(*
SPDX-FileCopyrightText: © 2026 Oleksandr Tiutyk <trofimich@gmail.com>
SPDX-License-Identifier: MIT
License: https://opensource.org/license/mit
*)

(*!
<summary>Stores an ordered sequence of generic values with fixed or dynamic capacity.</summary>
<description>
CreateEnumerator allocates an independent cursor owned by its caller. The collection must remain alive while
that cursor is used. Dynamic growth preserves the existing buffer on allocation failure and invokes the
terminal allocation-failure mechanism. Sort uses GENERIC_VALUE.CompareTo unless an explicit borrowed comparer
is supplied; descriptors preserve OBJECT and USER_DEFINED categories. Successful insertion transfers disposal
responsibility for owned payload; borrowed payload must remain alive while stored. The caller-side descriptor
copy is not reset and must not be released again after transfer. Independent owning aliases and overlapping
owned allocations are unsupported. Entries retain order and duplicates. Same-allocation replacement preserves
ownership without releasing retained storage. Get, FindSingle and enumerators only borrow payload.
ContainsGeneric defaults to releasing its query. Validators are borrowed for the collection lifetime. No
locking or mutation-version checks are implemented; callbacks that mutate the collection can invalidate
in-progress operations. Generic lookup with requested query release also attempts cleanup on lookup failure
before propagating the captured exception; terminal OOM takes precedence.
Instances cannot be assigned by value: copying backing pointers or disposal responsibility would create
unsafe aliases. Interface references still borrow this instance; copying an interface does not clone storage.
</description>
*)

{attribute 'no_explicit_call' := 'do not call this function block directly'}
FUNCTION_BLOCK List 
VAR_GENERIC CONSTANT
 	{attribute 'hide'} 
	//! <summary>Inline capacity; zero selects dynamic backing storage.</summary>
	_StaticCapacity : TOF_Core.DINT_LENGTH := 0;
END_VAR
EXTENDS TOF_Core.Object IMPLEMENTS IList
VAR_INPUT
	//! <summary>Number of slots added when dynamic storage is full; must be positive when growth is required.</summary>
	DefaultDynamicAllocationElementCount : BYTE := 10;	
END_VAR
VAR_STAT
	//! <summary>Class name shared by all instances of this function block.</summary>
	{attribute 'hide'} 
	_ClassName : STRING := __POUNAME();
END_VAR
VAR
	{attribute 'hide'} 
	_ValueValidator : TOF_Core.IGenericValueValidator;

	{attribute 'hide'} 
	_Array : POINTER TO TOF_Core.GENERIC_VALUE;
	{attribute 'hide'} 
	_StaticArray : ARRAY [0.._StaticCapacity - 1] OF TOF_Core.GENERIC_VALUE;
	
	{attribute 'hide'} 
	_DynamicCapacity : TOF_Core.DINT_LENGTH;
	{attribute 'hide'} 
	_Length : TOF_Core.DINT_LENGTH;
END_VAR

(*!
<summary>Grows the dynamic element buffer while preserving existing values.</summary>
<description>
Static instances return without allocation. A positive increment must fit DINT capacity and the UDINT
allocation-byte limit; invalid ranges raise ArgumentOutOfRangeException before storage changes. A null
allocation invokes the terminal allocation-failure mechanism before copying or deleting the old buffer.
Existing descriptors are moved without cloning payload; incoming ownership is not accepted by this helper.
Descendants cannot override this storage operation; capacity, indexing and disposal remain governed by this
collection implementation.
</description>
*)
METHOD PROTECTED FINAL AllocateMemory 
VAR_INPUT
	elementCount : TOF_Core.DINT_LENGTH;
END_VAR
VAR CONSTANT
	//! <summary>Bytes per capacity slot, including descriptor storage and any hash-index arrays.</summary>
	ENTRY_ALLOCATION_SIZE : ULINT := XSIZEOF(TOF_Core.GENERIC_VALUE);
END_VAR
VAR
	newMemory : POINTER TO TOF_Core.GENERIC_VALUE;
	newCapacity : ULINT;

END_VAR
IF NOT Dynamic THEN
	RETURN;
END_IF

IF elementCount <= TOF_Core.SignedInt32.ZERO THEN
	TOF_Core.Exceptions.ThrowArgumentOutOfRange(
		sourceNamespaceName := NamespaceName,
		sourceClassName := ClassName,
		sourcePOUName := __POUNAME(),
		sourcePosition := __POSITION(),
		argumentName := 'elementCount',
		argumentValue := elementCount
	);
END_IF

newCapacity := TO_ULINT(_DynamicCapacity) + TO_ULINT(elementCount);

IF newCapacity > TO_ULINT(TOF_Core.SignedInt32.MAX_VALUE)
	OR_ELSE newCapacity > TO_ULINT(TOF_Core.UnsignedInt32.MAX_VALUE) / ENTRY_ALLOCATION_SIZE
THEN
	TOF_Core.Exceptions.ThrowArgumentOutOfRange(
		sourceNamespaceName := NamespaceName,
		sourceClassName := ClassName,
		sourcePOUName := __POUNAME(),
		sourcePosition := __POSITION(),
		argumentName := 'capacity',
		argumentValue := newCapacity
	);
END_IF

newMemory := __NEW(BYTE, TO_UDINT(ENTRY_ALLOCATION_SIZE * newCapacity));

IF newMemory = 0 THEN
	TOF_Core.DynamicMemoryManager.RaiseAllocationFailure();
END_IF

IF _Length > TOF_Core.SignedInt32.ZERO THEN
	Tc2_System.MEMCPY(destAddr := newMemory, srcAddr := _Array, n := TO_UDINT(ENTRY_ALLOCATION_SIZE * TO_ULINT(_Length)));
END_IF

IF _Array <> 0 THEN
	__DELETE(_Array);
END_IF

_DynamicCapacity := TO_DINT(newCapacity);
_Array := newMemory;
END_METHOD

(*!
<summary>Copies a value and appends the owned descriptor.</summary>
<description>
Borrows the original during the call. isObject = TRUE requires a live Object FB instance implementing
ICloneable; other data is copied as bytes without recursively cloning references. A prepared copy is released
if insertion fails before acceptance; exceptions propagate. Engine-managed exception objects are unsupported.
index is meaningful only on success. Descendants cannot override this storage operation; capacity, indexing
and disposal remain governed by this collection implementation.
The original failure is captured before cleanup so nested cleanup handling cannot replace its payload.
A static native wrapper is cloned before cleanup; failure to capture still attempts prepared-copy disposal.
Terminal allocation failure takes precedence and no exception clone is allocated after its latch is set.
</description>
*)
METHOD FINAL AppendCopy : IList
VAR_INPUT
	value : ANY;
	isObject : BOOL := FALSE;
END_VAR
VAR_OUTPUT
	index : TOF_Core.DINT_INDEX;
END_VAR
VAR
	exceptionCode : __SYSTEM.ExceptionCode;
	caughtException : TOF_Core.IException;
	genericValue : TOF_Core.GENERIC_VALUE;
END_VAR

genericValue := TOF_Core.GenericValueFactory.FromAnyType(
		value := value,
		isObject := isObject,
		memoryManagementBehavior := TOF_Core.GENERIC_MEMORY_MANAGEMENT_BEHAVIOR.CLONE_ORIGINAL_VALUE_AND_OWNS_MEMORY
	);

__TRY
	AppendCopy := AppendGeneric(value := genericValue, index => index);
__CATCH(exceptionCode)
	caughtException := TOF_Core.ExceptionManager.GetLastException(
		exceptionCode := exceptionCode,
		catchPointNamespaceName := NamespaceName,
		catchPointPOUName := __POUNAME(),
		catchPointPosition := __POSITION()
	);
__ENDTRY

IF caughtException <> 0 THEN
	__TRY
		TOF_Core.DynamicMemoryManager.RaiseIfAllocationFailed();

		IF NOT caughtException.IsDynamicInstance THEN
			__QUERYINTERFACE(caughtException.Clone(), caughtException);
		END_IF
	__CATCH(exceptionCode)
		genericValue.Release();

		TOF_Core.ExceptionManager.ReThrowLastException(
			exceptionCode := exceptionCode,
			catchPointNamespaceName := NamespaceName,
			catchPointPOUName := __POUNAME(),
			catchPointPosition := __POSITION()
		);
	__ENDTRY

	genericValue.Release();

	TOF_Core.ExceptionManager.Throw(exception := caughtException);
END_IF
END_METHOD

(*!
<summary>Appends a descriptor to the list.</summary>
<description>
Successful insertion transfers disposal responsibility for owned payload; borrowed payload must remain alive
while stored. The caller-side descriptor copy is not reset and must not be released again after transfer.
Independent owning aliases and overlapping owned allocations are unsupported. Delegates to InsertGeneric;
index is meaningful only on success. Descendants cannot override this storage operation; capacity, indexing
and disposal remain governed by this collection implementation.
</description>
*)
METHOD FINAL AppendGeneric : IList
VAR_INPUT
	value : TOF_Core.GENERIC_VALUE;
END_VAR
VAR_OUTPUT
	index : TOF_Core.DINT_INDEX;
END_VAR
index := _Length;

AppendGeneric := InsertGeneric(index := index, value := value);
END_METHOD

(*!
<summary>Reports the currently allocated number of slots.</summary>
<description>
Units are bytes for ByteList and entries for other collections. Static capacity is fixed; dynamic capacity can
change on growth or clearing. This is not a guarantee that the next allocation succeeds.
</description>
*)
{attribute 'monitoring' := 'call'}
PROPERTY FINAL Capacity : TOF_Core.DINT_LENGTH
GET
Capacity := SEL(_StaticCapacity = 0, _StaticCapacity, _DynamicCapacity);
END_GET
END_PROPERTY

(*!
<summary>Borrows the concrete collection class name without transferring storage ownership.</summary>
*)
{attribute 'monitoring' := 'call'}
PROPERTY ClassName : REFERENCE TO STRING
GET
ClassName REF= _ClassName;
END_GET
END_PROPERTY

(*!
<summary>Removes all entries and releases dynamic backing storage.</summary>
<description>
Owned payload is released best effort through GENERIC_VALUE.Release; borrowed storage is not freed. Static
capacity and the borrowed validator are retained. Dynamic capacity becomes zero. Returns this collection and
invalidates positions and views. Cleanup callbacks must not reenter mutation. Descendants cannot override this
storage operation; capacity, indexing and disposal remain governed by this collection implementation.
</description>
*)
METHOD FINAL Clear : IList
VAR
	i : DINT;
END_VAR
Clear := THIS^;

FOR i := 0 TO _Length - 1 DO
	_Array[i].Release();						
END_FOR	

_Length := 0;
_DynamicCapacity := 0;

IF _Array <> 0 AND_THEN Dynamic THEN
	__DELETE(_Array);	
END_IF
END_METHOD

(*!
<summary>Searches for a value using default generic equality.</summary>
<description>
Borrows the ANY argument during a linear search without cloning or releasing it. isObject = TRUE means a live
Object FB instance, not a pointer or interface variable. Equality exceptions propagate; callbacks that mutate
the collection can invalidate traversal. Descendants cannot override this storage operation; capacity,
indexing and disposal remain governed by this collection implementation.
</description>
*)
METHOD FINAL Contains : BOOL
VAR_INPUT
	value : ANY;
	isObject : BOOL := FALSE;
END_VAR
VAR
	genericValue : TOF_Core.GENERIC_VALUE;
	i : TOF_Core.DINT_INDEX;
END_VAR

genericValue := TOF_Core.GenericValueFactory.FromAnyType(
		value := value,
		isObject := isObject,
		memoryManagementBehavior := TOF_Core.GENERIC_MEMORY_MANAGEMENT_BEHAVIOR.STORE_ORIGINAL_REFERENCE_AND_NOT_OWNS_MEMORY
	);

FOR i := 0 TO _Length - 1 DO
	IF _Array[i].Equals(otherValue := genericValue) THEN
		Contains := TRUE;
		RETURN;
	END_IF
END_FOR
END_METHOD

(*!
<summary>Searches for an equal generic value and optionally releases the query.</summary>
<description>
Uses GENERIC_VALUE.Equals in a linear search. releaseValue defaults to TRUE: after a completed search, Release
is called on the local query copy, including on a miss. Caller-side aliases are not reset. The query must not
own storage retained by the collection. Requested release is attempted after both successful lookup and lookup
failure. Before cleanup, the original framework exception is retained and a borrowed static system exception
is cloned to preserve its code, catch point and timestamps across cleanup callbacks. The captured exception is
then propagated through ExceptionManager.Throw in the current cyclic task; native errors use the framework
SystemException representation. If capturing the system exception fails with terminal OOM, query cleanup is
still attempted and terminal OOM takes precedence. Terminal allocation state is never cleared. Release is best
effort and does not prove successful deallocation. Cleanup callbacks must not reenter collection mutation.
Descendants cannot override this storage operation; capacity, indexing and disposal remain governed by this
collection implementation.
</description>
*)
METHOD FINAL ContainsGeneric : BOOL
VAR_INPUT
	value : TOF_Core.GENERIC_VALUE;
	releaseValue : BOOL := TRUE;
END_VAR
VAR
	exceptionCode : __SYSTEM.ExceptionCode;
	caughtException : TOF_Core.IException;

	i : DINT;
END_VAR
__TRY
	FOR i := 0 TO _Length - 1 DO
		IF _Array[i].Equals(otherValue := value) THEN
			ContainsGeneric := TRUE;
			EXIT;
		END_IF
	END_FOR
__CATCH(exceptionCode)
	caughtException := TOF_Core.ExceptionManager.GetLastException(
		exceptionCode := exceptionCode,
		catchPointNamespaceName := NamespaceName,
		catchPointPOUName := __POUNAME(),
		catchPointPosition := __POSITION()
	);
__ENDTRY

IF releaseValue THEN
	IF caughtException <> 0 AND_THEN NOT caughtException.IsDynamicInstance THEN
		__TRY
			TOF_Core.DynamicMemoryManager.RaiseIfAllocationFailed();
			__QUERYINTERFACE(caughtException.Clone(), caughtException);
		__CATCH(exceptionCode)
			value.Release();

			TOF_Core.ExceptionManager.ReThrowLastException(
				exceptionCode := exceptionCode,
				catchPointNamespaceName := NamespaceName,
				catchPointPOUName := __POUNAME(),
				catchPointPosition := __POSITION()
			);
		__ENDTRY
	END_IF

	value.Release();
END_IF

IF caughtException <> 0 THEN
	TOF_Core.ExceptionManager.Throw(exception := caughtException);
END_IF
END_METHOD

(*!
<summary>Creates an independent enumerator owned by the caller.</summary>
<description>
The caller must explicitly release the enumerator and keep this collection alive while using it. Allocation
failure invokes DynamicMemoryManager.RaiseAllocationFailure without a heap exception; it is terminal and is
not returned as a recoverable null result.
</description>
*)
METHOD CreateEnumerator : TOF_Core.IEnumerator
VAR
	enumerator : POINTER TO ListEnumerator;
END_VAR
enumerator := __NEW(ListEnumerator(list := THIS^));

IF enumerator = 0 THEN
	TOF_Core.DynamicMemoryManager.RaiseAllocationFailure();
END_IF

CreateEnumerator := enumerator^;
END_METHOD

(*!
<summary>Reports whether storage can grow dynamically.</summary>
<description>
Static capacity zero selects dynamic storage. Dynamic collections can still fail to allocate.
</description>
*)
{attribute 'monitoring' := 'call'}
PROPERTY FINAL Dynamic : BOOL
GET
Dynamic := _StaticCapacity = 0;
END_GET
END_PROPERTY

(*!
<summary>Reports whether the collection has no entries.</summary>
<description>
Reflects Length; not a check of payload lifetime or memory health.
</description>
*)
{attribute 'monitoring' := 'call'}
PROPERTY FINAL Empty : BOOL
GET
Empty := _Length <= 0;
END_GET
END_PROPERTY

(*!
<summary>Releases owned payload and backing storage during destruction.</summary>
<description>
Calls Clear; lifecycle methods and payload cleanup callbacks must not raise exceptions or reenter mutation.
Payload release is best effort, not proof of successful destruction. No separate copy-code ownership handoff
is implemented.
</description>
*)

METHOD FB_exit : BOOL
VAR_INPUT
	bInCopyCode : BOOL; 
END_VAR
Clear();
END_METHOD

(*!
<summary>Binds the optional validator and inline storage during initialization.</summary>
<description>
The validator is borrowed and must remain alive while used; it is not invoked here. Static storage is bound
without allocation. Lifecycle methods must not raise exceptions. No explicit online-change relocation repair
is implemented.
</description>
*)
METHOD FB_init : BOOL
VAR_INPUT
	bInitRetains : BOOL; // TRUE: the retain variables are initialized (reset warm / reset cold)
	bInCopyCode : BOOL; // TRUE: the instance will be copied to the copy code afterward (online change)
	valueValidator : TOF_Core.IGenericValueValidator;
END_VAR
_ValueValidator := valueValidator;

IF NOT Dynamic THEN
	_Array := ADR(_StaticArray); 
END_IF
END_METHOD

(*!
<summary>Finds a predicate match in the requested traversal direction.</summary>
<description>
skip counts matches, not visited entries. A null predicate or no match returns FALSE; outputs are meaningful
only on TRUE. The result is borrowed even if IsMemoryOwner is TRUE. Predicate input uses AsAnyType without
preserving the explicit generic OBJECT category. Predicate exceptions propagate; callbacks must not mutate the
traversed collection. Descendants cannot override this storage operation; capacity, indexing and disposal
remain governed by this collection implementation.
</description>
*)
METHOD FINAL FindSingle : BOOL
VAR_INPUT
	predicate : TOF_Core.IPredicate;
	skip : UDINT := 0;
	searchDirection : TOF_Core.SEARCH_DIRECTION := TOF_Core.SEARCH_DIRECTION.FROM_BEGINNING;
END_VAR
VAR_OUTPUT
	value : TOF_Core.GENERIC_VALUE;
	index : TOF_Core.DINT_INDEX;
END_VAR
VAR
	startSearchIndex : DINT;
	maxSearchIndex : DINT;
	indexStep : DINT;
	
	i : DINT;
	
	currentValue : __SYSTEM.AnyType;

	skippedMatchCount : UDINT := 0;
END_VAR
index := 0;
	
IF TO_DINT(skip) >= _Length OR_ELSE predicate = 0 THEN
	RETURN;
END_IF

startSearchIndex := SEL(searchDirection = TOF_Core.SEARCH_DIRECTION.FROM_BEGINNING, _Length - 1, 0);
maxSearchIndex := SEL(searchDirection = TOF_Core.SEARCH_DIRECTION.FROM_BEGINNING, 0, _Length - 1);
indexStep := SEL(searchDirection = TOF_Core.SEARCH_DIRECTION.FROM_BEGINNING, -1, 1);

FOR i := startSearchIndex TO maxSearchIndex BY indexStep DO
	currentValue := _Array[i].AsAnyType();
	
	IF predicate.Check(valueToCompare := currentValue) THEN
		IF skip = skippedMatchCount THEN
			value := _Array[i];
			index := i;
			FindSingle := TRUE;
			RETURN;
		ELSE
			skippedMatchCount := skippedMatchCount + 1;
		END_IF
	END_IF
END_FOR
END_METHOD

(*!
<summary>Reports whether fixed-capacity storage has no free slot.</summary>
<description>
Dynamic collections report FALSE even when Length equals Capacity. This does not guarantee available heap
memory.
</description>
*)
{attribute 'monitoring' := 'call'}
PROPERTY FINAL Full : BOOL
GET
Full := _StaticCapacity <> 0 AND_THEN _Length >= _StaticCapacity;
END_GET
END_PROPERTY

(*!
<summary>Borrows the descriptor at a zero-based list position.</summary>
<description>
An out-of-range index raises an exception. Returned descriptors and payload are borrowed, not clones. Do not
modify descriptor metadata or release payload through this view, even when IsMemoryOwner is TRUE. Keep the
source and borrowed storage alive; mutation or destruction can invalidate the view. Descendants cannot
override this storage operation; capacity, indexing and disposal remain governed by this collection
implementation.
</description>
*)
METHOD FINAL Get : REFERENCE TO TOF_Core.GENERIC_VALUE
VAR_INPUT
	index : TOF_Core.DINT_INDEX;
END_VAR
IF index < 0 OR_ELSE index >= _Length THEN
	TOF_Core.Exceptions.ThrowArgumentOutOfRange(
		sourceNamespaceName := NamespaceName,
		sourceClassName := ClassName,
		sourcePOUName := __POUNAME(),
		sourcePosition := __POSITION(),
		argumentName := 'index',
		argumentValue := index
	);
END_IF

Get REF= _Array[index];
END_METHOD

(*!
<summary>Copies a value and inserts it at the requested position.</summary>
<description>
Borrows the original during the call. isObject = TRUE requires a live Object FB instance implementing
ICloneable; other data is copied as bytes without recursively cloning references. A prepared copy is released
if insertion fails before acceptance; exceptions propagate. Engine-managed exception objects are unsupported.
The position may range from zero through Length inclusive. Descendants cannot override this storage operation;
capacity, indexing and disposal remain governed by this collection implementation.
The original failure is captured before cleanup so nested cleanup handling cannot replace its payload.
A static native wrapper is cloned before cleanup; failure to capture still attempts prepared-copy disposal.
Terminal allocation failure takes precedence and no exception clone is allocated after its latch is set.
</description>
*)
METHOD FINAL InsertCopy : IList
VAR_INPUT
	index : TOF_Core.DINT_INDEX;
	value : ANY;
	isObject : BOOL := FALSE;
END_VAR
VAR
	exceptionCode : __SYSTEM.ExceptionCode;
	caughtException : TOF_Core.IException;
	genericValue : TOF_Core.GENERIC_VALUE;
END_VAR

genericValue := TOF_Core.GenericValueFactory.FromAnyType(
		value := value,
		isObject := isObject,
		memoryManagementBehavior := TOF_Core.GENERIC_MEMORY_MANAGEMENT_BEHAVIOR.CLONE_ORIGINAL_VALUE_AND_OWNS_MEMORY
	);

__TRY
	InsertCopy := InsertGeneric(index := index, value := genericValue);
__CATCH(exceptionCode)
	caughtException := TOF_Core.ExceptionManager.GetLastException(
		exceptionCode := exceptionCode,
		catchPointNamespaceName := NamespaceName,
		catchPointPOUName := __POUNAME(),
		catchPointPosition := __POSITION()
	);
__ENDTRY

IF caughtException <> 0 THEN
	__TRY
		TOF_Core.DynamicMemoryManager.RaiseIfAllocationFailed();

		IF NOT caughtException.IsDynamicInstance THEN
			__QUERYINTERFACE(caughtException.Clone(), caughtException);
		END_IF
	__CATCH(exceptionCode)
		genericValue.Release();

		TOF_Core.ExceptionManager.ReThrowLastException(
			exceptionCode := exceptionCode,
			catchPointNamespaceName := NamespaceName,
			catchPointPOUName := __POUNAME(),
			catchPointPosition := __POSITION()
		);
	__ENDTRY

	genericValue.Release();

	TOF_Core.ExceptionManager.Throw(exception := caughtException);
END_IF
END_METHOD

(*!
<summary>Inserts a descriptor and shifts subsequent entries to the right.</summary>
<description>
Successful insertion transfers disposal responsibility for owned payload; borrowed payload must remain alive
while stored. The caller-side descriptor copy is not reset and must not be released again after transfer.
Independent owning aliases and overlapping owned allocations are unsupported. index may range from zero
through Length inclusive. Invalid indices and full static storage raise exceptions. Validation precedes
insertion. Dynamic growth rejects nonpositive increments and unrepresentable capacity or allocation sizes
before insertion. Descendants cannot override this storage operation; capacity, indexing and disposal remain
governed by this collection implementation.
</description>
*)
METHOD FINAL InsertGeneric : IList
VAR_INPUT
	index : TOF_Core.DINT_INDEX;
	value : TOF_Core.GENERIC_VALUE;	
END_VAR
VAR
	
	i : DINT;
END_VAR
IF index < 0 OR_ELSE index > _Length THEN
	TOF_Core.Exceptions.ThrowArgumentOutOfRange(
		sourceNamespaceName := NamespaceName,
		sourceClassName := ClassName,
		sourcePOUName := __POUNAME(),
		sourcePosition := __POSITION(),
		argumentName := 'index',
		argumentValue := index
	);
END_IF

IF _ValueValidator <> 0 THEN
	_ValueValidator.Validate(validatedObjectName := GetName(), valueToValidate := value);
END_IF

InsertGeneric := THIS^;

IF _Length >= Capacity THEN
	IF Dynamic THEN
		AllocateMemory(elementCount := DefaultDynamicAllocationElementCount);
	ELSE
		TOF_Core.Exceptions.ThrowStaticCollectionFull(
			sourceNamespaceName := NamespaceName,
			sourceClassName := ClassName,
			sourcePOUName := __POUNAME(),
			sourcePosition := __POSITION(),
			collectionName := GetName(),
			capacity := TO_UDINT(Capacity)
		);
	END_IF
END_IF

_Length := _Length + 1;

i := _Length - 1;

WHILE i > index DO
	_Array[i] := _Array[i - 1];	
	i := i - 1;
END_WHILE

_Array[i] := value;
END_METHOD

(*!
<summary>Reports the number of stored entries.</summary>
<description>
Units are bytes for ByteList and entries for other collections. Existing positions range from zero through
Length minus one.
</description>
*)
{attribute 'monitoring' := 'call'}
PROPERTY FINAL Length : TOF_Core.DINT_LENGTH
GET
Length := _Length;
END_GET
END_PROPERTY

(*!
<summary>Provides the library namespace for diagnostics.</summary>
<description>
Borrowed read-only reference to compiler-initialized metadata; no ownership transfer.
</description>
*)
{attribute 'monitoring' := 'call'}
PROPERTY NamespaceName : REFERENCE TO STRING
GET
NamespaceName REF= CurrentNamespace.Name;
END_GET
END_PROPERTY

(*!
<summary>Removes an existing list entry and compacts subsequent entries.</summary>
<description>
Invalid indices raise an exception. Owned payload is released best effort through GENERIC_VALUE.Release;
borrowed payload is not freed. Returns this list. Positions and descriptor references may change; cleanup
callbacks must not reenter mutation. Descendants cannot override this storage operation; capacity, indexing
and disposal remain governed by this collection implementation.
</description>
*)
METHOD FINAL RemoveAt : IList
VAR_INPUT
	index : TOF_Core.DINT_INDEX;
END_VAR
IF index < 0 OR_ELSE index >= _Length THEN
	TOF_Core.Exceptions.ThrowArgumentOutOfRange(
		sourceNamespaceName := NamespaceName,
		sourceClassName := ClassName,
		sourcePOUName := __POUNAME(),
		sourcePosition := __POSITION(),
		argumentName := 'index',
		argumentValue := index
	);
END_IF

RemoveAt := THIS^;

_Array[index].Release();			

IF index < _Length - 1 THEN
	Tc2_System.MEMMOVE(
		destAddr := ADR(_Array[index]),
		srcAddr := ADR(_Array[index + 1]),
		n := TO_UDINT(SIZEOF(TOF_Core.GENERIC_VALUE) * (_Length - index - 1))
	);
END_IF

_Array[_Length - 1].Reset();	

_Length := _Length - 1;
END_METHOD

(*!
<summary>Removes the first list entry equal to a borrowed query.</summary>
<description>
Uses default GENERIC_VALUE equality; isObject = TRUE requires a live Object FB instance. Reports removed on a
successful match and returns this list. Owned stored payload is released; the query is not adopted or
separately released. Equality exceptions propagate. Descendants cannot override this storage operation;
capacity, indexing and disposal remain governed by this collection implementation.
</description>
*)
METHOD FINAL RemoveFirst : IList
VAR_INPUT
	value : ANY;
	isObject : BOOL := FALSE;
END_VAR
VAR_OUTPUT
	removed : BOOL;
END_VAR
VAR
	genericValue : TOF_Core.GENERIC_VALUE;
	i : TOF_Core.DINT_INDEX;
END_VAR
RemoveFirst := THIS^;

IF _Length > 0 THEN
	genericValue := TOF_Core.GenericValueFactory.FromAnyType(
		value := value,
		isObject := isObject,
		memoryManagementBehavior := TOF_Core.GENERIC_MEMORY_MANAGEMENT_BEHAVIOR.STORE_ORIGINAL_REFERENCE_AND_NOT_OWNS_MEMORY
	);
	
	FOR i := 0 TO _Length - 1 DO
		IF _Array[i].Equals(otherValue := genericValue) THEN
			RemoveAt(index := i);
			removed := TRUE;
			RETURN;
		END_IF
	END_FOR
END_IF
END_METHOD

(*!
<summary>Removes predicate matches while traversing from the end.</summary>
<description>
skip counts matches from the end. A null predicate or maxRemoved = 0 performs no removal. Removes at most
maxRemoved matching entries after skipping the requested matches. Stops immediately after reaching the limit,
without invoking the predicate for remaining entries. Predicate exceptions propagate after any completed
removals, without rollback. removedCount counts completed removals. Callbacks must not mutate the traversed
collection. Descendants cannot override this storage operation; capacity, indexing and disposal remain
governed by this collection implementation.
</description>
*)
METHOD FINAL RemoveMatched : IList
VAR_INPUT
	predicate : TOF_Core.IPredicate;
	skip : UDINT := 0;
	maxRemoved : UDINT := TOF_Core.UnsignedInt32.MAX_VALUE;
END_VAR
VAR_OUTPUT
	removedCount : DINT;
END_VAR
VAR
	i : DINT;

	currentValue : __SYSTEM.AnyType;

	skippedMatchCount : UDINT := 0;
END_VAR
RemoveMatched := THIS^;

IF TO_DINT(skip) >= _Length OR_ELSE predicate = 0 OR_ELSE maxRemoved = TOF_Core.UnsignedInt32.MIN_VALUE THEN
	RETURN;
END_IF

FOR i := _Length - 1 TO 0 BY -1 DO
	currentValue := _Array[i].AsAnyType();
	
	IF predicate.Check(valueToCompare := currentValue) THEN
		IF skip <= skippedMatchCount THEN
			RemoveAt(index := i);
			removedCount := removedCount + 1;

			IF TO_UDINT(removedCount) >= maxRemoved THEN
				EXIT;
			END_IF
		ELSE
			skippedMatchCount := skippedMatchCount + 1;
		END_IF
	END_IF
END_FOR
END_METHOD

(*!
<summary>Restores the heap order below a root within the active sort range.</summary>
<description>
Requires valid indices and the same ordering selection used by Sort. A null comparer selects
GENERIC_VALUE.CompareTo; an explicit comparer takes precedence. Uses typed entry addresses and swaps
complete descriptors in place. Comparison exceptions propagate without rolling back completed swaps.
</description>
*)
METHOD PRIVATE restoreHeapFrom
VAR_INPUT
	rootIndex : DINT;
	heapSize : DINT;
	comparer : TOF_Core.IComparer;
	direction : TOF_Core.SORT_DIRECTION;
END_VAR
VAR
	currentIndex : DINT;
	childIndex : DINT;
	selectedIndex : DINT;

	comparisonResult : TOF_Core.COMPARISON_RESULT;

	value1, value2 : POINTER TO TOF_Core.GENERIC_VALUE;
END_VAR
currentIndex := rootIndex;

WHILE (currentIndex * 2 + 1) < heapSize DO
	childIndex := currentIndex * 2 + 1;
	selectedIndex := currentIndex;

	value1 := ADR(_Array[selectedIndex]);
	value2 := ADR(_Array[childIndex]);

	IF comparer = 0 THEN
		comparisonResult := value1^.CompareTo(otherValue := value2^);
	ELSE
		comparisonResult := comparer.Compare(first := value1^, second := value2^);
	END_IF

	IF direction = TOF_Core.SORT_DIRECTION.ASCENDING THEN
		IF comparisonResult = TOF_Core.COMPARISON_RESULT.FIRST_LESS_THAN_SECOND THEN
			selectedIndex := childIndex;
		END_IF
	ELSE
		IF comparisonResult = TOF_Core.COMPARISON_RESULT.FIRST_GREATER_THAN_SECOND THEN
			selectedIndex := childIndex;
		END_IF
	END_IF

	IF (childIndex + 1) < heapSize THEN
		value1 := ADR(_Array[selectedIndex]);
		value2 := ADR(_Array[childIndex + 1]);

		IF comparer = 0 THEN
			comparisonResult := value1^.CompareTo(otherValue := value2^);
		ELSE
			comparisonResult := comparer.Compare(first := value1^, second := value2^);
		END_IF

		IF direction = TOF_Core.SORT_DIRECTION.ASCENDING THEN
			IF comparisonResult = TOF_Core.COMPARISON_RESULT.FIRST_LESS_THAN_SECOND THEN
				selectedIndex := childIndex + 1;
			END_IF
		ELSE
			IF comparisonResult = TOF_Core.COMPARISON_RESULT.FIRST_GREATER_THAN_SECOND THEN
				selectedIndex := childIndex + 1;
			END_IF
		END_IF
	END_IF

	IF selectedIndex = currentIndex THEN
		RETURN;
	END_IF

	Swap(index1 := currentIndex, index2 := selectedIndex);
	
	currentIndex := selectedIndex;
END_WHILE
END_METHOD

(*!
<summary>Reports the size of this function-block instance.</summary>
<description>
Measured in bytes; includes inline storage but excludes separately allocated buffers, payload and enumerators.
</description>
*)
{attribute 'monitoring' := 'call'}
PROPERTY SelfSize : ULINT
GET
SelfSize := XSIZEOF(THIS^);
END_GET
END_PROPERTY

(*!
<summary>Copies a value and stores it through SetGeneric.</summary>
<description>
Borrows the original during the call. isObject = TRUE requires a live Object FB instance implementing
ICloneable; other data is copied as bytes without recursively cloning references. A prepared copy is released
if insertion fails before acceptance; exceptions propagate. Engine-managed exception objects are unsupported.
Any index output is meaningful only on success. Descendants cannot override this storage operation; capacity,
indexing and disposal remain governed by this collection implementation.
The original failure is captured before cleanup so nested cleanup handling cannot replace its payload.
A static native wrapper is cloned before cleanup; failure to capture still attempts prepared-copy disposal.
Terminal allocation failure takes precedence and no exception clone is allocated after its latch is set.
</description>
*)
METHOD FINAL SetCopy : IList
VAR_INPUT
	index : TOF_Core.DINT_INDEX;
	value : ANY;
	isObject : BOOL := FALSE;
END_VAR
VAR
	exceptionCode : __SYSTEM.ExceptionCode;
	caughtException : TOF_Core.IException;
	genericValue : TOF_Core.GENERIC_VALUE;
END_VAR

genericValue := TOF_Core.GenericValueFactory.FromAnyType(
		value := value,
		isObject := isObject,
		memoryManagementBehavior := TOF_Core.GENERIC_MEMORY_MANAGEMENT_BEHAVIOR.CLONE_ORIGINAL_VALUE_AND_OWNS_MEMORY
	);

__TRY
	SetCopy := SetGeneric(index := index, value := genericValue);
__CATCH(exceptionCode)
	caughtException := TOF_Core.ExceptionManager.GetLastException(
		exceptionCode := exceptionCode,
		catchPointNamespaceName := NamespaceName,
		catchPointPOUName := __POUNAME(),
		catchPointPosition := __POSITION()
	);
__ENDTRY

IF caughtException <> 0 THEN
	__TRY
		TOF_Core.DynamicMemoryManager.RaiseIfAllocationFailed();

		IF NOT caughtException.IsDynamicInstance THEN
			__QUERYINTERFACE(caughtException.Clone(), caughtException);
		END_IF
	__CATCH(exceptionCode)
		genericValue.Release();

		TOF_Core.ExceptionManager.ReThrowLastException(
			exceptionCode := exceptionCode,
			catchPointNamespaceName := NamespaceName,
			catchPointPOUName := __POUNAME(),
			catchPointPosition := __POSITION()
		);
	__ENDTRY

	genericValue.Release();

	TOF_Core.ExceptionManager.Throw(exception := caughtException);
END_IF
END_METHOD

(*!
<summary>Replaces the descriptor at an existing list position.</summary>
<description>
Successful replacement transfers disposal responsibility for owned payload; borrowed payload must remain alive
while stored. The caller-side descriptor copy is not reset and must not be released again after transfer.
Invalid indices and rejected validation raise exceptions before replacement. Reusing the same allocation
preserves existing ownership or accepts incoming ownership without releasing that allocation. Aliases must
have compatible disposal semantics; independently owned aliases and overlapping owned ranges are unsupported.
A different displaced allocation is released best effort after installing the new descriptor. Cleanup
callbacks must not reenter collection mutation. Descendants cannot override this storage operation; capacity,
indexing and disposal remain governed by this collection implementation.
</description>
*)
METHOD FINAL SetGeneric : IList
VAR_INPUT
	index : TOF_Core.DINT_INDEX;
	value : TOF_Core.GENERIC_VALUE;	
END_VAR
VAR

	displacedValue : TOF_Core.GENERIC_VALUE;
END_VAR
IF index < TOF_Core.SignedInt32.ZERO OR_ELSE index >= _Length THEN
	TOF_Core.Exceptions.ThrowArgumentOutOfRange(
		sourceNamespaceName := NamespaceName,
		sourceClassName := ClassName,
		sourcePOUName := __POUNAME(),
		sourcePosition := __POSITION(),
		argumentName := 'index',
		argumentValue := index
	);
END_IF

IF _ValueValidator <> 0 THEN
	_ValueValidator.Validate(validatedObjectName := GetName(), valueToValidate := value);
END_IF

SetGeneric := THIS^;

displacedValue := _Array[index];

IF displacedValue.Address = value.Address THEN
	IF displacedValue.IsMemoryOwner AND_THEN NOT value.IsMemoryOwner THEN
		value := TOF_Core.GenericValueFactory.FromParts(
			genericTypeClass := value.TypeClass,
			address := value.Address,
			size := value.Size,
			memoryManagementBehavior := TOF_Core.GENERIC_MEMORY_MANAGEMENT_BEHAVIOR.STORE_ORIGINAL_REFERENCE_AND_OWNS_MEMORY
		);
	END_IF

	displacedValue.Reset();
END_IF

_Array[index] := value;
displacedValue.Release();
END_METHOD

(*!
<summary>Reorders entries in place using the supplied generic-value ordering strategy.</summary>
<description>
A null or omitted comparer selects GENERIC_VALUE.CompareTo for each pair. An explicit comparer takes
precedence and must provide a consistent order for the stored representations. Payload and comparer are
borrowed. The default order supports Core numeric, text, temporal and OBJECT comparison rules; incompatible
pairs raise GenericConversionNotSupportedException and OBJECT values require IComparable. Empty and singleton
lists return without invoking comparisons. Callbacks must not modify operands or the collection. Exceptions
propagate without rolling back completed swaps; every descriptor and its ownership remain in the list.
Returns this list. Descendants cannot override the storage operation.
</description>
*)
//!<param name="comparer">Optional borrowed ordering strategy; zero selects GENERIC_VALUE.CompareTo.</param>
//!<param name="direction">Requested ordering direction.</param>
METHOD FINAL Sort : IList
VAR_INPUT
	comparer : TOF_Core.IComparer := 0;
	direction : TOF_Core.SORT_DIRECTION := TOF_Core.SORT_DIRECTION.ASCENDING;
END_VAR
VAR CONSTANT
	//! <summary>Largest entry count using insertion sort; larger lists use in-place heap sort.</summary>
	SMALL_LIST_SORT_LIMIT : DINT := 16;
END_VAR
VAR

	i : DINT;
	j : DINT;
	startIndex : DINT;
	endIndex : DINT;

	comparisonResult : TOF_Core.COMPARISON_RESULT;

	value1, value2 : TOF_Core.GENERIC_VALUE;
END_VAR
Sort := THIS^;

IF _Length <= 1 THEN
	RETURN;
END_IF

// Insertion sort is faster for small lists, otherwise use heap sort
IF _Length <= SMALL_LIST_SORT_LIMIT THEN
	FOR i := 1 TO _Length - 1 DO
		j := i;

		WHILE j > 0 DO
			value1 := _Array[j - 1];
			value2 := _Array[j];

			IF comparer = 0 THEN
				comparisonResult := value1.CompareTo(otherValue := value2);
			ELSE
				comparisonResult := comparer.Compare(first := value1, second := value2);
			END_IF

			IF direction = TOF_Core.SORT_DIRECTION.ASCENDING THEN
				IF comparisonResult <> TOF_Core.COMPARISON_RESULT.FIRST_GREATER_THAN_SECOND THEN
					EXIT;
				END_IF
			ELSE
				IF comparisonResult <> TOF_Core.COMPARISON_RESULT.FIRST_LESS_THAN_SECOND THEN
					EXIT;
				END_IF
			END_IF

			Swap(index1 := j - 1, index2 := j);
			
			j := j - 1;
		END_WHILE
	END_FOR

	RETURN;
END_IF

// Build heap
startIndex := (_Length / 2) - 1;

WHILE startIndex >= 0 DO
	restoreHeapFrom(rootIndex := startIndex, heapSize := _Length, comparer := comparer, direction := direction);
	
	startIndex := startIndex - 1;
END_WHILE

// Extract heap root into the final sorted position
endIndex := _Length - 1;

WHILE endIndex > 0 DO
	Swap(index1 := 0, index2 := endIndex);
	
	restoreHeapFrom(rootIndex := 0, heapSize := endIndex, comparer := comparer, direction := direction);
	
	endIndex := endIndex - 1;
END_WHILE
END_METHOD

(*!
<summary>Exchanges two positions without cloning or releasing payload.</summary>
<description>
Returns this list. Different indices must be valid or an exception is raised. Current implementation returns
immediately for equal indices without validating them. Payload ownership is preserved. Descendants cannot
override this storage operation; capacity, indexing and disposal remain governed by this collection
implementation.
</description>
*)
METHOD FINAL Swap : IList
VAR_INPUT
	index1 : TOF_Core.DINT_INDEX;
	index2 : TOF_Core.DINT_INDEX;
END_VAR
VAR
	tmp : TOF_Core.GENERIC_VALUE;
END_VAR
Swap := THIS^;

IF index1 = index2 THEN
	RETURN;
ELSIF index1 < 0 OR_ELSE index1 >= _Length THEN
	TOF_Core.Exceptions.ThrowArgumentOutOfRange(
		sourceNamespaceName := NamespaceName,
		sourceClassName := ClassName,
		sourcePOUName := __POUNAME(),
		sourcePosition := __POSITION(),
		argumentName := 'index1',
		argumentValue := index1
	);
ELSIF index2 < 0 OR_ELSE index2 >= _Length THEN
	TOF_Core.Exceptions.ThrowArgumentOutOfRange(
		sourceNamespaceName := NamespaceName,
		sourceClassName := ClassName,
		sourcePOUName := __POUNAME(),
		sourcePosition := __POSITION(),
		argumentName := 'index2',
		argumentValue := index2
	);
END_IF

tmp := _Array[index1];
_Array[index1] := _Array[index2];
_Array[index2] := tmp;
END_METHOD

(*!
<summary>Exposes the configured value validator.</summary>
<description>
Borrowed optional reference fixed at initialization. Zero means no validator. The collection does not own or
release it.
</description>
*)
{attribute 'monitoring' := 'call'}
PROPERTY FINAL ValueValidator : TOF_Core.IGenericValueValidator
GET
ValueValidator := _ValueValidator;
END_GET
END_PROPERTY

END_FUNCTION_BLOCK

(* stored: Version 1.1.0.1
   POU List: Id {423efb90-4c6a-41e3-8889-647ff943b33e}, SpecialFunc None
   Folder Service methods: Id {3188279f-4192-4144-9219-d1281be18b24}
   Method AllocateMemory: Id {7805ad4a-1088-4228-99dd-d8b7fe4579c3}
   Method AppendCopy: Id {c48f84f5-3206-4f8e-a06b-95fdd5877efa}
   Method AppendGeneric: Id {f1ff6a71-50a0-45d9-ae86-164a44b67bf8}
   Property Capacity: Id {f88ebbc6-043e-4384-9aab-efeb366abd1b}
   Get Get: Id {e0e73894-ad23-446a-99c0-aacf7f854d6b}
   Property ClassName: Id {33e07dae-fed5-4e1d-8f43-eee6214a3816}
   Get Get: Id {f6501ffd-91a8-433d-945c-613d26b30c47}
   Method Clear: Id {6eeb2dd8-b2fb-4bd3-af28-3d4655f329b4}
   Method Contains: Id {6470b115-1732-45d7-86e6-432cfb852dab}
   Method ContainsGeneric: Id {4f27da2f-dece-43c4-8992-282ab34ccb18}
   Method CreateEnumerator: Id {9c229dd9-393b-46ff-976f-739fe26eedc5}
   Property Dynamic: Id {166b951e-511c-4d32-bb47-240a0b602e17}
   Get Get: Id {629e79ca-4190-4ac7-928c-69e20f8bf579}
   Property Empty: Id {6c336543-2ac9-4adb-b317-6015c15c963c}
   Get Get: Id {cbbea261-31d9-4fda-a46a-9b7d9838e2ea}
   Method FB_exit: Id {8d8b7b19-3218-490a-a08e-e708f6895db1}
   Method FB_init: Id {7bc30a89-0227-48d6-bfc1-e831cfff4350}
   Method FindSingle: Id {5bd8df97-f8f3-46ed-97e0-2baa71205501}
   Property Full: Id {142088f9-89b6-4514-9bf8-182d44bd5096}
   Get Get: Id {60f38d2d-7d5e-4f53-bd6e-39eabf1a5689}
   Method Get: Id {35156606-e33f-4fd7-a3f8-50e4c6feea06}
   Method InsertCopy: Id {7c5e7ea9-1602-45c2-9555-47aa08559820}
   Method InsertGeneric: Id {2dcf43ab-5d4d-40f0-ba4f-54f191c32509}
   Property Length: Id {8b78c4a9-2b51-4df9-a89b-35d75f4063d7}
   Get Get: Id {40434b4f-ac59-4ed2-adb0-38a6ead17ebd}
   Property NamespaceName: Id {790d2c44-7c10-4ff7-8e9f-92d4936a4655}
   Get Get: Id {dfd8ff83-c535-4eea-abbd-5a05ac36fe99}
   Method RemoveAt: Id {0e28301b-e63b-49ca-a697-ef9528fc2481}
   Method RemoveFirst: Id {ab28382f-e74f-44a6-bee2-f905f3030356}
   Method RemoveMatched: Id {e5cc38ae-8b20-4e35-acc9-fcd84e9d10bd}
   Method restoreHeapFrom: Id {1a1c5c77-8af0-4f17-a539-272de7e4b0a4}
   Property SelfSize: Id {b8f1c23e-6bde-4d17-b77f-f3d1373a6f6b}
   Get Get: Id {0c60dbce-56ff-4644-ae28-c3c705772b31}
   Method SetCopy: Id {e9638d43-e88c-48cb-a07f-937c5e87c232}
   Method SetGeneric: Id {28fb4746-7d53-4b08-a432-54d437f989bb}
   Method Sort: Id {cd2a8a15-72bb-44f7-9e5d-ecb76fed56a8}
   Method Swap: Id {eb0e8297-edd7-472f-a573-82e2ae740339}
   Property ValueValidator: Id {b948083e-197f-42c4-870d-0ac963bd346a}
   Get Get: Id {cb2fa504-489a-4e73-8b3c-20c2650b6edd} *)
